RoboDK station: ME5286_Lab4_Azamat_Turganbayev.rdk

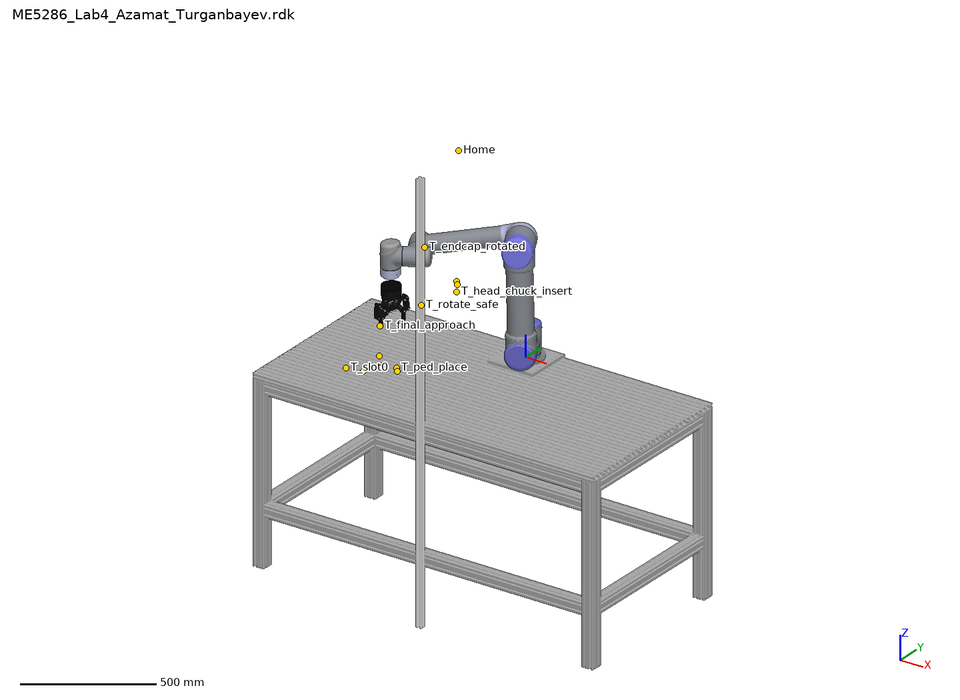
[picture v0: the station drawn from its stored meshes, robots at their saved joint values, targets as dots, program paths as lines]
Station ur5_and_table_and_gripper_spring26 (saved by RoboDK 5.9.6). Poses are relative to the parent item; angles as X-Y-Z fixed-axis rotations.
  - frame UR5 Base at (0, 0, 0) mm
    - robot UR5: 6 axes, payload 5 kg, reach 850 mm, repeatability 0.1 mm, weight 18.4 kg
        modified DH rows (alpha deg, a mm, theta deg, d mm): 0, 0, 0, 89.2; 90, 0, 180, 0; 0, 425, 0, 0; 0, 392.43, 0, 109; -90, 0, 0, 93.65; 90, 0, 180, 82
        joint limits [-360, -360, -360, -360, -360, -360] to [360, 360, 360, 360, 360, 360]; home [0, -90, 90, 0, 90, 0]; saved at [27.777, -88.789, 99.606, -99.203, -89.492, 225.953]
      - tool Gripper RobotiQ 85 Opened, TCP at (0, 0, 211.5) mm, size 147.4 x 146.8 x 75 mm
      - tool W-010-B_20200218, TCP at (0, 0, 150) mm, size 75 x 75 x 16.9 mm, geometry from W-010-B_20200218.STEP
      - object ROBOTIQ_FTS-300-SEN-001_20181119_20210810 at (0, 0, 0) mm, size 120.4 x 191.7 x 37.2 mm, geometry from ROBOTIQ_FTS-300-SEN-001_20181119_20210810.STEP
    - target Home (joint target) at (-17.73, -403.36, 999.72) mm, rotated rx -90 ry 2 rz -178 deg; joints [2, -88, 0, -90, 0, 0] of UR5
    - target T_ped_place (Cartesian target) at (-260.43, -455.65, 66.5) mm, rotated rx 87.71 ry 2.06 rz -97.78 deg; joints [80.793, -58.719, 120.622, -118.564, -182.744, 301.307] of UR5
    - target T_slot0 (Cartesian target) at (-484.06, -458.04, 3.09) mm, rotated rx 175.55 ry -1.96 rz 91.28 deg; joints [33.678, -58.164, 80.144, -107.173, -89.268, 32.445] of UR5
    - target T_rotate_safe (Cartesian target) at (-227.41, -344.97, 286.66) mm, rotated rx 179.27 ry -3.39 rz 92.4 deg; joints [42.853, -98.571, 87.601, -76.27, -92.103, 40.529] of UR5
    - target T_endcap_rotated (Cartesian target) at (-202.98, -356.11, 535.47) mm, rotated rx 91.41 ry -0.5 rz -92.67 deg; joints [87.054, -106.217, 102.301, -97.549, -178.559, 259.031] of UR5
    - target T_slot2 (Cartesian target) at (-328.9, -459.64, 57.19) mm, rotated rx 175.82 ry 0.46 rz 98.8 deg; joints [41.882, -75, 96.607, -108.357, -87.337, 32.986] of UR5
    - target T_slot1 (Cartesian target) at (-406.08, -456.73, 12.56) mm, rotated rx 179.26 ry -1.89 rz 92.29 deg; joints [38.616, -67.169, 93.199, -114.31, -91.088, 36.354] of UR5
    - target T_chuck_approach (Cartesian target) at (-332.34, 32.32, 342.78) mm, rotated rx 176.36 ry -3.15 rz 75.63 deg; joints [-21.327, -106.5, 84.997, -65.254, -93.561, -6.752] of UR5
    - target T_head_chuck_insert (Cartesian target) at (-332.64, 32.06, 160.98) mm, rotated rx 176.35 ry -3.12 rz 75.54 deg; joints [-21.301, -110.18, 114.467, -91.028, -93.522, -6.641] of UR5
    - target T_batt_insert (Cartesian target) at (-333.66, 36.25, 202.06) mm, rotated rx 174.52 ry -3.36 rz 85.44 deg; joints [-20.823, -109.066, 107.618, -84.217, -94.744, -15.924] of UR5
    - target T_endcap_thread_press (Cartesian target) at (-330.93, 35.42, 190.15) mm, rotated rx 177.21 ry -1.45 rz 73.2 deg; joints [-23.583, -111.416, 111.036, -87.017, -91.77, -6.705] of UR5
    - target T_flash_pick (Cartesian target) at (-332.64, 32.06, 160.98) mm, rotated rx 176.35 ry -3.12 rz 75.54 deg; joints [-21.301, -110.18, 114.467, -91.028, -93.522, -6.641] of UR5
    - target T_ped_pick (Cartesian target) at (-253.37, -458.19, 55.22) mm, rotated rx -179.37 ry 2.28 rz 176.96 deg; joints [47.797, -81.567, 105.562, -113.045, -87.833, 320.832] of UR5
    - target T_endcap_twist_1 (Cartesian target) at (-331.01, 36.44, 189.58) mm, rotated rx 179.99 ry 0.42 rz 67.91 deg; joints [-25.781, -113.863, 113.094, -89.193, -89.579, 356.311] of UR5
    - target T_final (Cartesian target) at (-334.26, -459.37, 96.63) mm, rotated rx 179.2 ry 1.46 rz 136.85 deg; joints [42.166, -77.597, 94.298, -105.788, -88.612, -4.708] of UR5
    - target T_final_approach (Cartesian target) at (-334.21, -456.78, 216.63) mm, rotated rx 179.2 ry 1.46 rz 136.92 deg; joints [41.97, -80.162, 79.642, -88.559, -88.612, -4.966] of UR5
  - object table_base_setup at (0, 0, 0) mm, rotated rx 0 ry 0 rz -90 deg, size 1524 x 762 x 800.1 mm, geometry from table_base_setup.STEP
  - object 6ft_beam_table at (0, -675, 1000) mm, size 25.4 x 25.4 x 1828.8 mm, geometry from 6ft_beam_table.IGS
  - Python program final (listed below)

--- Python program final ---
from robodk.robolink import *
from robodk.robomath import *

RDK = Robolink()
robot = RDK.Item('', ITEM_TYPE_ROBOT)

# All targets
HOME         = RDK.Item('Home')
T_SLOT0      = RDK.Item('T_slot0')                          # endcap pickup pose
T_SLOT1      = RDK.Item('T_slot1')                          # battery pickup at tray slot 1
T_SLOT2      = RDK.Item('T_slot2')                          # head pickup at tray slot 2
T_SLOT3      = RDK.Item('T_ped_place')                      # placement of endcap at tray slot 3
T_ROT_SAFE   = RDK.Item('T_rotate_safe')                    # safe pose to begin endcap rotation
T_ENDCAP_ROT = RDK.Item('T_endcap_rotated')                 # endcap rotation
T_CHUCK_APP  = RDK.Item('T_chuck_approach')                 # safe above chuck
T_HEAD_INS   = RDK.Item('T_head_chuck_insert')              # head seated in chuck
T_BATT_INS   = RDK.Item('T_batt_insert')                    # battery aligned above head opening
T_PED_PICK   = RDK.Item('T_ped_pick')                       # pickup the endcap from pedestal
T_ENDCAP_THREAD_PRESS = RDK.Item('T_endcap_thread_press')   # endcap on the head
T_ENDCAP_TWIST_1   = RDK.Item('T_endcap_twist_1')           # endcap rotation
T_FINAL_APP = RDK.Item('T_final_approach')                  # approach slot 2
T_FINAL = RDK.Item('T_final')                               # final pose


# Tunables
CLEAR_Z = 100   # mm for leaving the poses
SPEED   = 600    # mm/s
ACCEL   = 700   # mm/s^2


robot.setSpeed(SPEED)
robot.setAcceleration(ACCEL)

def set_default_speed():
    robot.setSpeedJoints(80)
    robot.setAccelerationJoints(150)


INSTR = INSTRUCTION_CALL_PROGRAM # for gripper
AUX_INSTR = INSTRUCTION_INSERT_CODE # for chuck

# Gripper functions

def gripper_open():
    robot.RunCodeCustom('rq_set_speed_norm(50)', INSTR)
    robot.RunCodeCustom('rq_open_and_wait()', INSTR)

def gripper_close():
    robot.RunCodeCustom('rq_set_force(50)', INSTR)
    robot.RunCodeCustom('rq_close_and_wait()', INSTR)

#  Leave target using Linear Movement

def moveL_Leave(target_item, dz_clear=CLEAR_Z):
    base = target_item.Pose()
    robot.MoveL(base * transl(0, 0, -dz_clear))

#  Leave target using Joint Movement

def moveJ_Leave(target_item, dz_clear=CLEAR_Z):
    base = target_item.Pose()
    robot.MoveJ(base * transl(0, 0, -dz_clear))

# Ensures not touching the objects during the movement

def moveJ_drop_leave_approach(target_item, dz_clear=CLEAR_Z):
    base = target_item.Pose()
    robot.MoveJ(base * transl(0, dz_clear, 0))

# Pick part from the target

def goto_pick(target_item):
    robot.MoveJ(target_item)
    gripper_close()
    moveL_Leave(target_item)

#place part to the target

def goto_place(target_item):
    robot.MoveJ(target_item)
    gripper_open()
    moveJ_drop_leave_approach(target_item)

#  Chuck functions

def clamp():
    robot.RunCodeCustom('clamp()', AUX_INSTR)

def unclamp():
    robot.RunCodeCustom('unclamp()', AUX_INSTR)

# Performs action of putting head of battery in the chuck

def put_head_in_chuck():
    moveJ_drop_leave_approach(T_SLOT3,300) # move safely from pedestal
    goto_pick(T_SLOT2)              # pick head from slot 2
    robot.MoveJ(T_CHUCK_APP)        # move above chuck
    moveJ_Leave(T_HEAD_INS, dz_clear = -5)
    gripper_open()                  # release head
    clamp()
    robot.MoveJ(T_CHUCK_APP)        # back out

# Performs action of putting battery in the flashlight head

def put_battery_in_head():
    goto_pick(T_SLOT1)              # pick battery from slot 1
    robot.MoveJ(T_CHUCK_APP)
    robot.MoveL(T_BATT_INS)         # align above opening
    gripper_open()
    robot.MoveJ(T_CHUCK_APP)

# Putting endcap on the flashlight head to begin the threading

def put_endcap_in_head():
    goto_pick(T_PED_PICK)
    robot.MoveJ(T_CHUCK_APP)
    robot.MoveJ(T_ENDCAP_THREAD_PRESS)

# Function for threading

def prethread_4_strokes():
    for _ in range(4):
        robot.setSpeedJoints(110)
        robot.setAccelerationJoints(170)
        gripper_close() # clamp endcap in gripper
        robot.MoveJ(T_ENDCAP_TWIST_1) # tightening stroke
        robot.RunCodeCustom('rq_move_and_wait_norm(50)', INSTRUCTION_INSERT_CODE) # slight open (regrip)
        robot.MoveJ(T_ENDCAP_THREAD_PRESS) # reset back to start pose

# Built in function

def final_tighten():
    robot.RunCodeCustom('tighten_torque(2, 0, 1.57, 2, 2, 1, 100, 100, 50)',INSTRUCTION_INSERT_CODE)

# action of placing the final assembly

def unload_and_return_to_slot2():
    gripper_open()
    gripper_close()
    unclamp()
    robot.MoveJ(T_CHUCK_APP)
    robot.MoveJ(T_FINAL_APP)
    robot.setSpeed(30)
    robot.setAcceleration(70)
    robot.MoveL(T_FINAL)
    gripper_open()
    robot.MoveL(T_FINAL_APP)


# Step 1 (Endcap)

robot.MoveJ(HOME)      # Start Home
set_default_speed()
gripper_open()

goto_pick(T_SLOT0)     # Pick endcap from slot 0
robot.MoveJ(T_ROT_SAFE)
robot.MoveJ(T_ENDCAP_ROT)
goto_place(T_SLOT3)    # Place on pedestal slot 3

# STEP 2 (head + battery)
put_head_in_chuck()
put_battery_in_head()

# STEP 3 (Endcap threading)
put_endcap_in_head()
robot.setRounding(-1) # ensures that it won't find the fastest approach to the T_ENDCAP_TWIST_1
prethread_4_strokes()
final_tighten()
set_default_speed()
unload_and_return_to_slot2()

robot.MoveJ(HOME)      # End Home
